// TIA Portal V18 export
TYPE "UDT_AnalogProxyCH_Vars"
// stored: IsFailsafeCompliant false
   STRUCT
      cCHModeCtrl : Array[1..8] of Byte;   // 0-Not Active, 1-StraigntSignal,2-Adapt , 3-NewSignal
      xCHRlyIsOnInd : Array[1..8] of Bool;   // Off/On
      xCHRlyIsOffInd : Array[1..8] of Bool;   // Off/On
      xCHRlyOnCmd : Array[1..8] of Bool;   // Off/On
      xCHRlyIndError : Array[1..8] of Bool;   // Norm/Alarm
      rCHDrivenSignal : Array[1..8] of Real;   // 0-100.0%
      rCHProxySignal : Array[1..8] of Real;   // 0-100.0%
   END_STRUCT;
END_TYPE
